// TIA Portal V20 export
DATA_BLOCK "MeasuringInput_FeedingRollAxisB_Tab"   // DB36, Motion_DB
// stored: InstanceOfName TO_MeasuringInput, OfSystemLibElement TO_MeasuringInput, OfSystemLibVersion 9.0
TO_MeasuringInput   // technology object, version 9.0
// stored: Connection Interface MeasuringInput, InputAddress 26400
   // // inherited from TO_Object
   // VAR
   //    Status { ExternalWritable := 'False'} : DInt;
   //    InputState { ExternalWritable := 'False'} : Bool;
   //    Parameter { S7_SetPoint := 'True'} : TO_MeasuringInput_Struct_Parameter;
   //    Interface { ExternalWritable := 'False'; S7_SetPoint := 'True'} : TO_MeasuringInput_Struct_Interface;
   //    MeasuredValues { ExternalWritable := 'False'; S7_SetPoint := 'True'} : TO_MeasuringInput_Struct_MeasuredValues;
   //    Units { ExternalWritable := 'False'; S7_SetPoint := 'True'} : TO_MeasuringInput_Struct_Units;
   //    StatusWord { ExternalWritable := 'False'} : DWord;
   //    ErrorWord { ExternalWritable := 'False'} : DWord;
   //    ErrorDetail { ExternalWritable := 'False'; S7_SetPoint := 'True'} : TO_Struct_ErrorDetail;
   //    WarningWord { ExternalWritable := 'False'} : DWord;
   // END_VAR
BEGIN
   Parameter.MeasuringRangeActivationTime := 40.0;
   Parameter.CorrectionTime := 0.23;
   Interface.Address.RID := 16#2000001;
   Interface.Address.AREA := 16#81;
   Interface.Address.OFFSET := 26400;
END_DATA_BLOCK
